// TIA Portal V20 export
TYPE "LBP_typeModularMcpBaseInput"
TITLE = Modular MCP image / Image MCP modulaire
// Input image of base signals for modular MCP / Image des entrées des signaux de base pour MCP modulaires
   STRUCT
      optionalKey1 : Bool;   // input image n+0 bit 0; KT-IN1 / Image des entrées n+0 bit 0 ; KT-IN1
      optionalKey2 : Bool;   // input image n+0 bit 1; KT-IN2 / Image des entrées n+0 bit 1 ; KT-IN2
      optionalKey3 : Bool;   // input image n+0 bit 2; KT-IN3 / Image des entrées n+0 bit 2 ; KT-IN3
      optionalKey4 : Bool;   // input image n+0 bit 3; KT-IN4 / Image des entrées n+0 bit 3 ; KT-IN4
      optionalKey5 : Bool;   // input image n+0 bit 4; KT-IN5 / Image des entrées n+0 bit 4 ; KT-IN5
      optionalKey6 : Bool;   // input image n+0 bit 5; KT-IN6 / Image des entrées n+0 bit 5 ; KT-IN6
      optionalKey7 : Bool;   // input image n+0 bit 6; KT-IN7 / Image des entrées n+0 bit 6 ; KT-IN7
      optionalKey8 : Bool;   // input image n+0 bit 7; KT-IN8 / Image des entrées n+0 bit 7 ; KT-IN8
      optionalKey9 : Bool;   // input image n+1 bit 0; KT-IN9 / Image des entrées n+1 bit 0 ; KT-IN9
      optionalKey10 : Bool;   // input image n+1 bit 1; KT-IN10 / Image des entrées n+1 bit 1 ; KT-IN10
      optionalKey11 : Bool;   // input image n+1 bit 2; KT-IN11 / Image des entrées n+1 bit 2 ; KT-IN11
      optionalKey12 : Bool;   // input image n+1 bit 3; KT-IN12 / Image des entrées n+1 bit 3 ; KT-IN12
      optionalKey13 : Bool;   // input image n+1 bit 4; KT-IN13 / Image des entrées n+1 bit 4 ; KT-IN13
      optionalKey14 : Bool;   // input image n+1 bit 5; KT-IN14 / Image des entrées n+1 bit 5 ; KT-IN14
      optionalKey15 : Bool;   // input image n+1 bit 6; KT-IN15 / Image des entrées n+1 bit 6 ; KT-IN15
      optionalKey16 : Bool;   // input image n+1 bit 7; KT-IN16 / Image des entrées n+1 bit 7 ; KT-IN16
      spindleOvr : USInt;   // input image byte n+2 / Image des entrées octet n+2
      feedrateOvr : USInt;   // input image byte n+3 / Image des entrées octet n+3
      keySwitch0 : Bool;   // input image n+4 bit 0 / Image des entrées n+4 bit 0
      keySwitch1 : Bool;   // input image n+4 bit 1 / Image des entrées n+4 bit 1
      keySwitch2 : Bool;   // input image n+4 bit 2 / Image des entrées n+4 bit 2
      keySwitch3 : Bool;   // input image n+4 bit 3 / Image des entrées n+4 bit 3
      reserved44 : Bool;
      reserved45 : Bool;
      reserved46 : Bool;
      reserved47 : Bool;
      reserved50 : Bool;
      reserved51 : Bool;
      reserved52 : Bool;
      reserved53 : Bool;
      reserved54 : Bool;
      reserved55 : Bool;
      reserved56 : Bool;
      reserved57 : Bool;
   END_STRUCT;
END_TYPE
